(* IEC 61131-3 sources: plcc/crates/plcc-cli/tests/data/image, 3 files *)

(* ---- chase.st ---- *)
(* SPDX-License-Identifier: MPL-2.0
   Program-image test (tests/image.rs): a TON-timed chase over three relays
   while %IX0.0 is on; the time comes from plcc_monotonic_ns, a service. *)
PROGRAM Chase
VAR
    t : TON;
    step : INT;
    run AT %IX0.0 : BOOL;
    r1 AT %QX0.0 : BOOL;
    r2 AT %QX0.1 : BOOL;
    r3 AT %QX0.2 : BOOL;
END_VAR
t(IN := run AND NOT t.Q, PT := T#100ms);
IF t.Q THEN
    step := (step + 1) MOD 3;
END_IF
r1 := run AND step = 0;
r2 := run AND step = 1;
r3 := run AND step = 2;
END_PROGRAM

(* ---- div_zero.st ---- *)
(* SPDX-License-Identifier: MPL-2.0
   Program-image test (tests/image.rs): a division by zero on the third scan
   must reach the runtime's plcc_fault service, not the object's weak default. *)
PROGRAM Div
VAR
    a : INT := 10;
    b : INT := 0;
    c AT %MW0 : INT;
    n AT %MW1 : INT;
END_VAR
n := n + 1;
IF n >= 3 THEN
    c := a / b;
END_IF
END_PROGRAM

(* ---- services.st ---- *)
(* SPDX-License-Identifier: MPL-2.0
   Program-image test (tests/image.rs): exercises runtime services through the
   veneers (64-bit division, libm, 64-bit <-> float conversions, plcc_print)
   and leaves the results in %M for the test to check. *)
PROGRAM Svc
VAR
    q AT %ML1 : LINT;
    r AT %ML2 : LINT;
    s AT %ML3 : LREAL;
    f AT %MD8 : REAL;
    g AT %MD9 : REAL;
    big AT %ML5 : LINT;
    n : LINT := 1234567890123;
    d : LINT := 1000;
    x : LREAL := 0.5;
    y : REAL := 0.25;
    done : BOOL;
END_VAR
IF NOT done THEN
    q := n / d;
    r := n MOD d;
    s := SIN(x) + EXPT(x, 2.5);
    f := LINT_TO_REAL(n);
    g := COS(y);
    big := n * 3;
    PRINT('services ok');
    done := TRUE;
END_IF
END_PROGRAM
